// TwinCAT 3 PLC project PLC_Student
// ProgramVersion: 3.1.4024.0
// libraries:
//   Tc2_Standard, * (Beckhoff Automation GmbH)
//   Tc2_System, * (Beckhoff Automation GmbH)
//   Tc3_Module, * (Beckhoff Automation GmbH)
//   VisuSymbols,3.5.10.0,System
// project tree:
//   / GlobalTextList.TcGTLO, PlcTask.TcTTO, Visualization Manager.TcVMO (not stored)
//   GVLs/ GVL.TcGVL
//   POUs/ Auto.TcPOU, MAIN.TcPOU, Manual.TcPOU (unreadable), TextDisplay.TcPOU
//   VISUs/ HMIControl.TcVIS

CONFIGURATION PLC_Student
    RESOURCE PLC ON TwinCAT3
        TASK PlcTask(INTERVAL := T#10ms, PRIORITY := 21);
        PROGRAM MAIN WITH PlcTask : MAIN;
    END_RESOURCE
END_CONFIGURATION

// ---- GVLs/GVL.TcGVL
{attribute 'qualified_only'}
VAR_GLOBAL
	// Input to PLC from process 
	ixSensor1		AT %I*: BOOL;		(* Sensor at First Station  *)
	ixSensor2		AT %I*: BOOL;		(* Sensor at Second Station *)
	
	qxButtRight		AT %Q*: BOOL;		(* Button for moving the tram Right *)
	qxButtLeft		AT %Q*: BOOL;		(* Button for moving the tram Left *)
	
	qxButtManual	AT %Q*: BOOL;		(* Button for Manual Mode *)
	qxButtAuto		AT %Q*: BOOL;		(* Button for Auto Mode *)
	
	qxButtEmerg     AT %Q*: BOOL;		(* Button for Emergency Stop *)
	
	mxManualRight   AT %Q*: BOOL;
	mxManualLeft    AT %Q*: BOOL;
	
	mxAutoRight     AT %Q*: BOOL;
	mxAutoLeft      AT %Q*: BOOL;
	
	mxEmergRight    AT %Q*: BOOL;
	mxEmergLeft     AT %Q*: BOOL;
	
	mxEmergManLeft  AT %Q*: BOOL;
	
END_VAR

// ---- POUs/MAIN.TcPOU
PROGRAM MAIN
VAR
END_VAR

Manual();
Auto();
TextDisplay();

END_PROGRAM

// ---- POUs/Auto.TcPOU
PROGRAM Auto
VAR
	MovRightS: BOOL;
	MovRightL: BOOL;
	MovLeftS: BOOL;
	TON_Right: TON;
	TON_Left: TON;
	
	Home: BOOL;
	HomeMemory: BOOL;
	ManRequest: BOOL;
	TON_Right1: TON;
	TON_Left1: TON;
END_VAR
VAR // added by the converter: edge detectors and wires of the graphical bodies
    _w1 : BOOL;
END_VAR

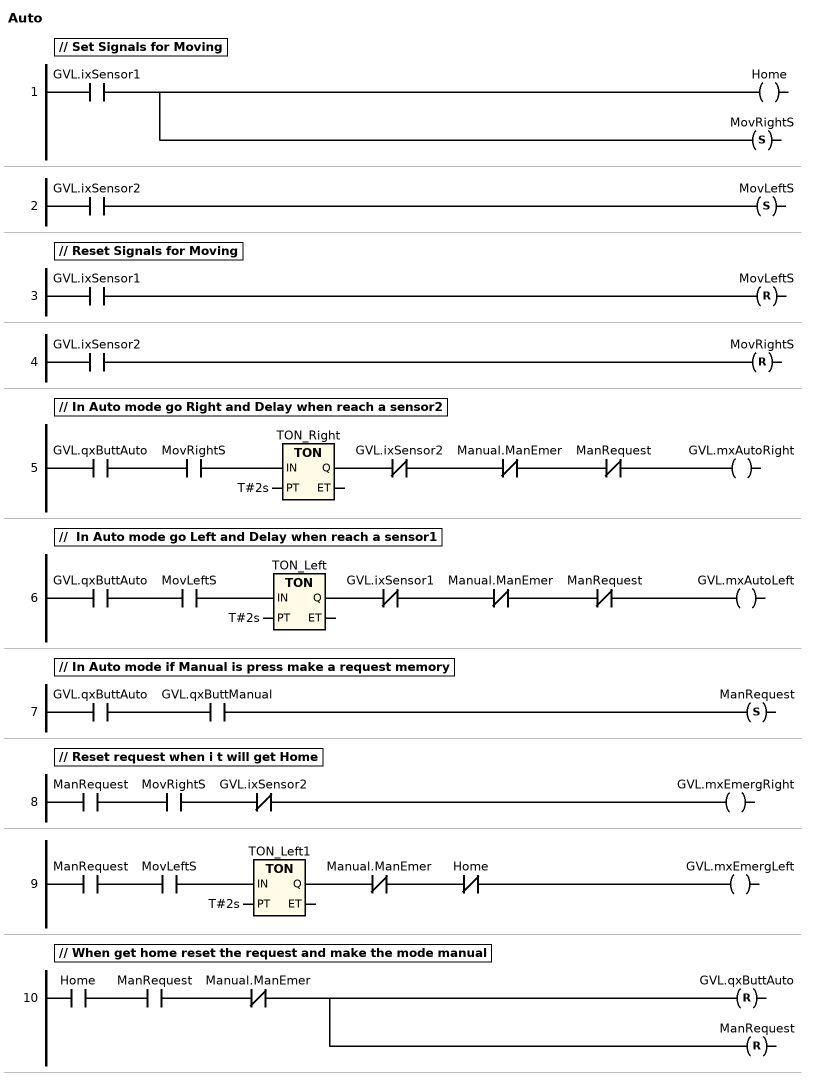
// NETWORK 1
// label: // Set Signals for Moving
Home := GVL.ixSensor1;
MovRightS S= GVL.ixSensor1;

// NETWORK 2
MovLeftS S= GVL.ixSensor2;

// NETWORK 3
// label: // Reset Signals for Moving
MovLeftS R= GVL.ixSensor1;

// NETWORK 4
MovRightS R= GVL.ixSensor2;

// NETWORK 5
// label: // In Auto mode go Right and Delay when reach a sensor2
TON_Right(IN := GVL.qxButtAuto AND MovRightS, PT := T#2s); // TON
GVL.mxAutoRight := TON_Right.Q AND NOT GVL.ixSensor2 AND NOT Manual.ManEmer AND NOT ManRequest;

// NETWORK 6
// label: //  In Auto mode go Left and Delay when reach a sensor1
TON_Left(IN := GVL.qxButtAuto AND MovLeftS, PT := T#2s); // TON
GVL.mxAutoLeft := TON_Left.Q AND NOT GVL.ixSensor1 AND NOT Manual.ManEmer AND NOT ManRequest;

// NETWORK 7
// label: // In Auto mode if Manual is press make a request memory
ManRequest S= GVL.qxButtAuto AND GVL.qxButtManual;

// NETWORK 8
// label: // Reset request when i t will get Home
GVL.mxEmergRight := ManRequest AND MovRightS AND NOT GVL.ixSensor2;

// NETWORK 9
TON_Left1(IN := ManRequest AND MovLeftS, PT := T#2s); // TON
GVL.mxEmergLeft := TON_Left1.Q AND NOT Manual.ManEmer AND NOT Home;

// NETWORK 10
// label: // When get home reset the request and make the mode manual
_w1 := Home AND ManRequest AND NOT Manual.ManEmer;
GVL.qxButtAuto R= _w1;
ManRequest R= _w1;

END_PROGRAM

// ---- POUs/TextDisplay.TcPOU
PROGRAM TextDisplay
VAR
	TextDis: STRING;
END_VAR

IF GVL.ixSensor1 THEN
	TextDis := 'Home';
ELSIF
	GVL.ixSensor2 THEN
	TextDis := 'Station 1';
ELSIF GVL.qxButtEmerg AND NOT GVL.qxButtRight AND NOT GVL.qxButtLeft THEN
	TextDis := 'Emergency Stop';
ELSE
	TextDis := 'Moving';
END_IF

END_PROGRAM

// ---- GlobalTextList.TcGTLO
TEXTLIST GlobalTextList
  236 = '%s'
  603 = '%s TextDisplay.TextDis'
  271 = '%TextDisplay.TextDis'
  373 = 'Auto'
  551 = 'Display'
  622 = 'E - Stop'
  656 = 'Emergency'
  644 = 'Emergency Button'
  183 = 'Manual'
  959 = 'TextDisplay.TextDis'
END_TEXTLIST

// ---- VISUs/HMIControl.TcVIS
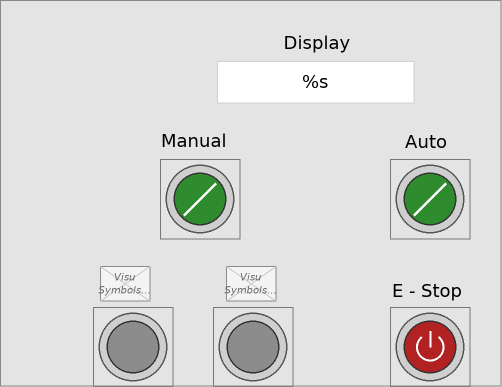
VISUALIZATION HMIControl  // 502x387
    Image (226,266 50x35), image: VisuSymbols.Symbols.ArrowBoldRight
    PushSwitch (88,307 90x80), variable: GVL.qxButtLeft, behaviour: TAP, style: Switch-PushSwitch-Gray
    PushSwitch (208,307 90x80), variable: GVL.qxButtRight, behaviour: TAP, style: Switch-PushSwitch-Gray
    Image (100,266 50x35), image: VisuSymbols.Symbols.ArrowBoldLeft
    Label (119,126 150x30), "Manual"
    RotarySwitch (155,159 90x80), variable: GVL.qxButtManual, behaviour: TOGGLE, style: Switch-RotarySwitch-Green
    RotarySwitch (385,159 90x80), variable: GVL.qxButtAuto, input disabled if: NOT Auto.Home, behaviour: TOGGLE, style: Switch-RotarySwitch-Green
    Label (351,127 150x30), "Auto"
    PowerSwitch (385,307 90x80), variable: GVL.qxButtEmerg, behaviour: TOGGLE, style: Switch-PowerSwitch-Red
    Label (352,276 150x30), "E - Stop"
    Textfield (217,61 197x42), "%s", text variable: TextDisplay.TextDis
    Label (242,28 150x30), "Display"
END_VISUALIZATION
